Omron CX-Programmer project 新工程 (CX-Programmer 9.73)

# PLC 新PLC1: CPM1(CPM1A) CPU30

## Program 新程序1 (no task)
; 本项目是为木材加工厂设计的自动化控制系统，旨在实现木材的高效、安全接合。 / 系统涉及的物理设备包括启动按钮、停止按钮、模式切换按钮、进料传感器、出料传感器、安全门开关、故障复位按钮、紧急停止按钮、进料电机、出料电机、主电机、辅助电机、加热器、冷却器、进料阀门、出料阀门、报警灯、运行指示灯、进料指示灯、出料指示灯。 / [计划实施] / 1.系统通过启动按钮激活系统使能。 / i.启动按钮按下时，系统进入准备状态。 / 2.操作员通过模式切换按钮选择运行模式，控制系统状态。 / 3.在自动模式下，进料电机和出料电机根据系统状态运行。 / 4.安全门开关打开时，进料电机停止，以防止意外伤害。 / 5.主电机在重置状态和冷却状态准备好且无故障状态时运行。 / i.主电机运行时，表示接合部件正常工作。 / ii.重置状态激活时，系统准备启动主电机。 / iii.冷却状态表示冷却过程完成。 / 6.加热器在模式切换按钮触发且辅助电机支持时运行。 / i.辅助电机运行时，支持加热器工作。 / ii.加热状态未激活时，允许加热器启动。 / 7.冷却器通过定时器控制冷却过程，如进料延时15秒、加热时间25秒。 / 8.运行状态根据停止按钮和进料电机状态调整，当停止按钮按下或进料电机停止时更新为停止。 / i.运行状态激活时，系统处于正常操作。 / ii.停止按钮用于暂停系统运行。 / 9.紧急停止按钮按下时，激活紧急停止状态，暂停系统操作。 / 10.故障状态在故障复位按钮按下、出料电机停止且定时器 TIM013 计时完成后清除。 / 11.在手动模式下，手动模式按钮启用操作员控制功能，通过自动模式按钮切换状态。 / 12.木材离开系统时，出料指示灯点亮。 / 13.系统配备运行指示灯、进料指示灯等状态指示，确保操作员了解设备状态。

### Section 段1

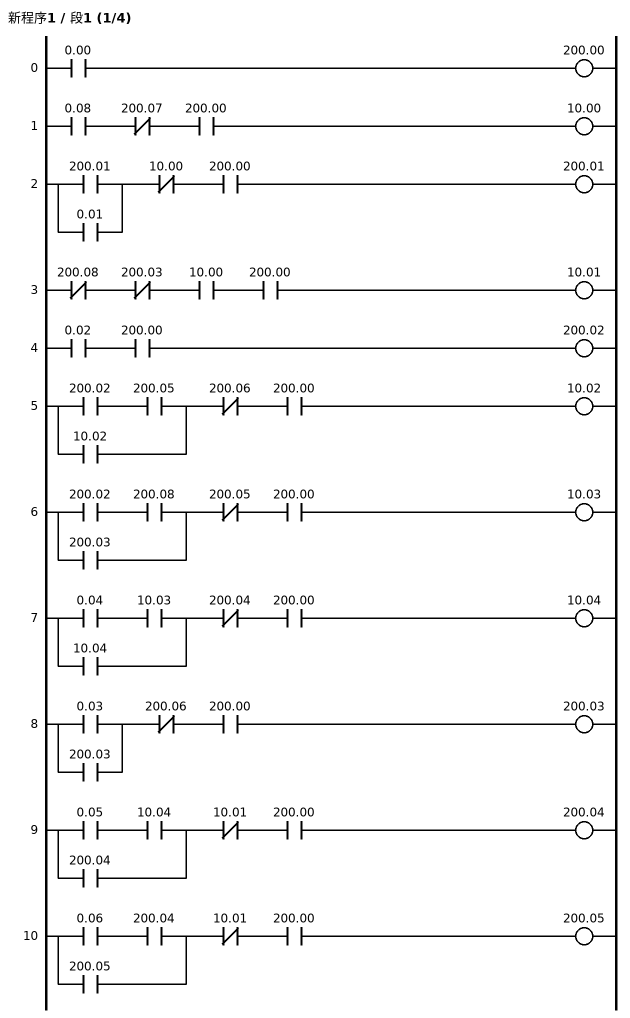
; rung 0
LD 0.00
OUT 200.00
; rung 1
LD 0.08
ANDNOT 200.07
AND 200.00
OUT 10.00
; rung 2
LD 200.01
OR 0.01
ANDNOT 10.00
AND 200.00
OUT 200.01
; rung 3
LDNOT 200.08
ANDNOT 200.03
AND 10.00
AND 200.00
OUT 10.01
; rung 4
LD 0.02
AND 200.00
OUT 200.02
; rung 5
LD 200.02
AND 200.05
OR 10.02
ANDNOT 200.06
AND 200.00
OUT 10.02
; rung 6
LD 200.02
AND 200.08
OR 200.03
ANDNOT 200.05
AND 200.00
OUT 10.03
; rung 7
LD 0.04
AND 10.03
OR 10.04
ANDNOT 200.04
AND 200.00
OUT 10.04
; rung 8
LD 0.03
OR 200.03
ANDNOT 200.06
AND 200.00
OUT 200.03
; rung 9
LD 0.05
AND 10.04
OR 200.04
ANDNOT 10.01
AND 200.00
OUT 200.04
; rung 10
LD 0.06
AND 200.04
OR 200.05
ANDNOT 10.01
AND 200.00
OUT 200.05

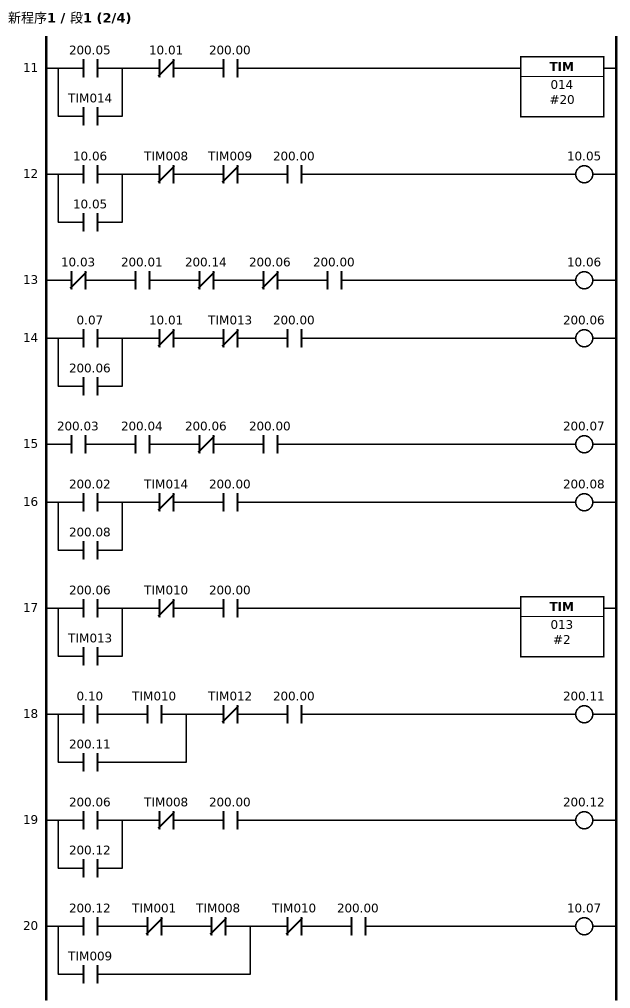
; rung 11
LD 200.05
OR TIM014
ANDNOT 10.01
AND 200.00
TIM 014 #20
; rung 12
LD 10.06
OR 10.05
ANDNOT TIM008
ANDNOT TIM009
AND 200.00
OUT 10.05
; rung 13
LDNOT 10.03
AND 200.01
ANDNOT 200.14
ANDNOT 200.06
AND 200.00
OUT 10.06
; rung 14
LD 0.07
OR 200.06
ANDNOT 10.01
ANDNOT TIM013
AND 200.00
OUT 200.06
; rung 15
LD 200.03
AND 200.04
ANDNOT 200.06
AND 200.00
OUT 200.07
; rung 16
LD 200.02
OR 200.08
ANDNOT TIM014
AND 200.00
OUT 200.08
; rung 17
LD 200.06
OR TIM013
ANDNOT TIM010
AND 200.00
TIM 013 #2
; rung 18
LD 0.10
AND TIM010
OR 200.11
ANDNOT TIM012
AND 200.00
OUT 200.11
; rung 19
LD 200.06
OR 200.12
ANDNOT TIM008
AND 200.00
OUT 200.12
; rung 20
LD 200.12
ANDNOT TIM001
ANDNOT TIM008
OR TIM009
ANDNOT TIM010
AND 200.00
OUT 10.07

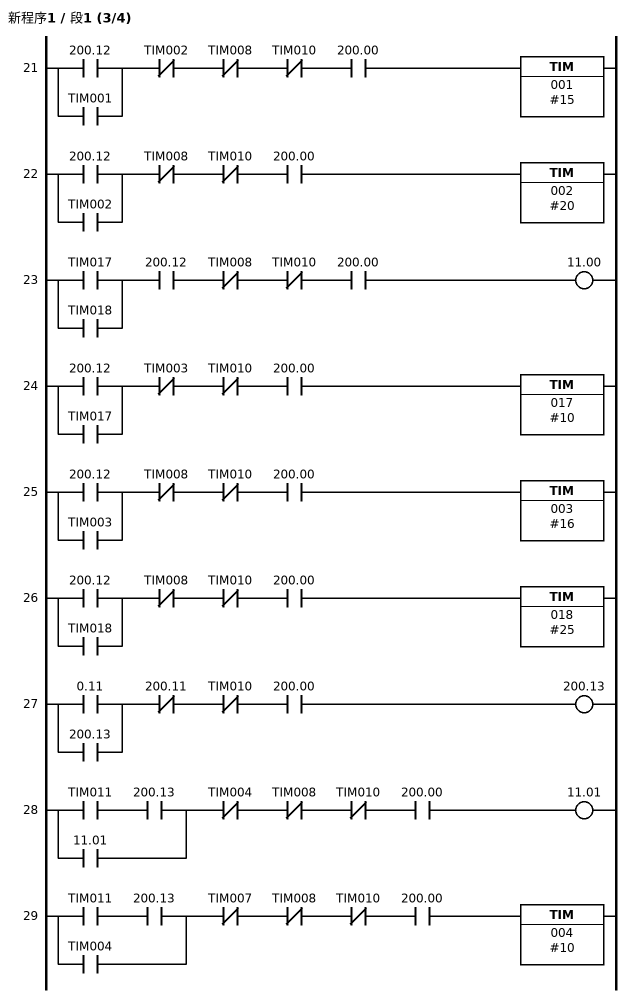
; rung 21
LD 200.12
OR TIM001
ANDNOT TIM002
ANDNOT TIM008
ANDNOT TIM010
AND 200.00
TIM 001 #15
; rung 22
LD 200.12
OR TIM002
ANDNOT TIM008
ANDNOT TIM010
AND 200.00
TIM 002 #20
; rung 23
LD TIM017
OR TIM018
AND 200.12
ANDNOT TIM008
ANDNOT TIM010
AND 200.00
OUT 11.00
; rung 24
LD 200.12
OR TIM017
ANDNOT TIM003
ANDNOT TIM010
AND 200.00
TIM 017 #10
; rung 25
LD 200.12
OR TIM003
ANDNOT TIM008
ANDNOT TIM010
AND 200.00
TIM 003 #16
; rung 26
LD 200.12
OR TIM018
ANDNOT TIM008
ANDNOT TIM010
AND 200.00
TIM 018 #25
; rung 27
LD 0.11
OR 200.13
ANDNOT 200.11
ANDNOT TIM010
AND 200.00
OUT 200.13
; rung 28
LD TIM011
AND 200.13
OR 11.01
ANDNOT TIM004
ANDNOT TIM008
ANDNOT TIM010
AND 200.00
OUT 11.01
; rung 29
LD TIM011
AND 200.13
OR TIM004
ANDNOT TIM007
ANDNOT TIM008
ANDNOT TIM010
AND 200.00
TIM 004 #10

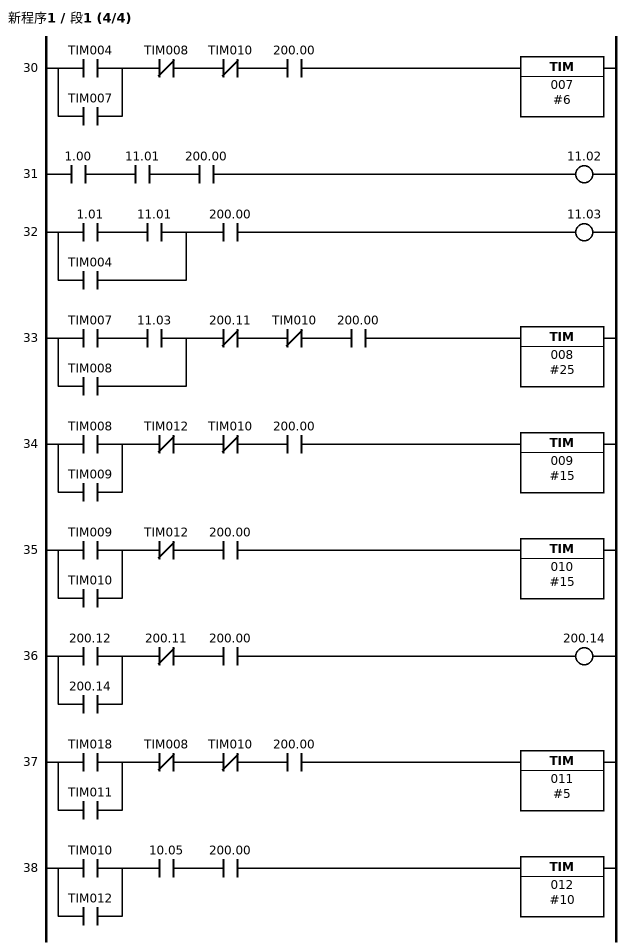
; rung 30
LD TIM004
OR TIM007
ANDNOT TIM008
ANDNOT TIM010
AND 200.00
TIM 007 #6
; rung 31
LD 1.00
AND 11.01
AND 200.00
OUT 11.02
; rung 32
LD 1.01
AND 11.01
OR TIM004
AND 200.00
OUT 11.03
; rung 33
LD TIM007
AND 11.03
OR TIM008
ANDNOT 200.11
ANDNOT TIM010
AND 200.00
TIM 008 #25
; rung 34
LD TIM008
OR TIM009
ANDNOT TIM012
ANDNOT TIM010
AND 200.00
TIM 009 #15
; rung 35
LD TIM009
OR TIM010
ANDNOT TIM012
AND 200.00
TIM 010 #15
; rung 36
LD 200.12
OR 200.14
ANDNOT 200.11
AND 200.00
OUT 200.14
; rung 37
LD TIM018
OR TIM011
ANDNOT TIM008
ANDNOT TIM010
AND 200.00
TIM 011 #5
; rung 38
LD TIM010
OR TIM012
AND 10.05
AND 200.00
TIM 012 #10
; rung 39
END(01)